FUNCTION_BLOCK FB_AdsCommunicationRead
VAR_INPUT
	NETID											: T_AmsNetID;
	AdsPORT											: T_AmsPort;
	IDXGRP											: UDINT;
	IDXOFFS											: UDINT;	
	TMOUT											: TIME;
END_VAR
VAR_OUTPUT
	bBusy											: BOOL;
	iBusyNumber 									: INT;
	bError											: BOOL;
	iErrorNumber									: INT;
	udiErrorID										: UDINT;
	stAdsCommunicationReadOUT						: ST_Communication;
END_VAR
VAR
	fbAdsCommunicationRead							: ADSREAD;			//Odczyt zmiennych 
	fbAdsReadStatus									: ADSRDSTATE;		//Odczyt stanu urządzenia ADS
	ftRead											: F_TRIG;
	bRead											: BOOL;	
	rtBusy											: R_TRIG;
	rtError											: R_TRIG;
	tonRefresh										: TON;
	udiErrorNumberTest: UDINT;
END_VAR


IF NOT bBusy AND NOT bError THEN
	bRead				:= TRUE;
END_IF
IF bError AND bRead THEN
	bRead				:= FALSE;
END_IF

ACT_AdsRead();

IF bError AND NOT bRead THEN
	bRead				:= TRUE;
END_IF

IF bRead AND NOT bError THEN
	bRead				:= FALSE;
END_IF

ACT_AdsRead();

rtBusy(CLK := bBusy);
rtError(CLK := bError);

IF rtBusy.Q THEN
    iBusyNumber                                                := iBusyNumber + 1;
    IF iBusyNumber = 32760 THEN
        iBusyNumber                                            := 0;
    END_IF
END_IF

IF rtError.Q THEN
    iErrorNumber                                                := iErrorNumber + 1;
    IF iErrorNumber = 32760 THEN
        iErrorNumber                                            := 0;
    END_IF
END_IF

IF NOT bError THEN
;	
ELSE
	;
END_IF


IF bError THEN
	udiErrorNumberTest		:= fbAdsCommunicationRead.ERRID;
END_IF

ACTION ACT_AdsRead:


fbAdsCommunicationRead(
	NETID:= 				NETID, 
	PORT:= 					AdsPORT, 
	IDXGRP:= 				IDXGRP, 
	IDXOFFS:= 				IDXOFFS, 
	LEN:= 					SIZEOF(stAdsCommunicationReadOUT), 
	DESTADDR:= 				ADR(stAdsCommunicationReadOUT), 
	READ:= 					bRead, 
	TMOUT:= 				TMOUT, 
	BUSY=> 					bBusy, 
	ERR=> 					bError, 
	ERRID=> 				udiErrorID);
END_ACTION

END_FUNCTION_BLOCK

(* stored: Version 1.1.0.1, ProductVersion 3.1.4026.13, FileIdentifier 560566f24c9706101f6fa783f44c16e4c7cc399c, FileSignature 2ac096a45061f9bae4ef418e5954f3c45b58cb6e839a9db37d6836598bb014766ce69df650efcef6209caad90ca48592432c34702bdbe991b569298511ceb36202963cdfa54cf538daaa3269a8950c9e3eb51f11993fd34bcfade7c4049b6efc442b884a8899dd6e364d3918dd11c09d345ead7ae2ce8d30e73fa0ea13537837ddc02c88108cf00255d530c57f8070067b6358bd11aa05834e850c8098d28bd44952c4443b7d51e9743dd8d0c33a175d83c9dd9d2a85fdc0dafe683c6c04b0e9bff6ec0d2d0e1aba34d8fbc6d7c104d0fefb94b7cc190db4eb4a32f291f521b0a4d719545a1194140cd90dacf3c79530a2fe9710404329fbb778bd441f2abc0f
   POU FB_AdsCommunicationRead: Id {af7872f0-b209-428e-9975-6fa9e5430ade}, SpecialFunc None
   Action ACT_AdsRead: Id {f3388244-206e-48af-a906-46ac44c69c17} *)
